% RSLogix 500 project 7.1.RSS, saved by version 8.30.00.16 %
PROJECT "UNTITLED"    % processor: Bul.1763 MicroLogix 1100 Series B %

PROGRAM FILES
  LAD 2   4 rungs

DATA FILES
  O0 OUTPUT  4 elements
  I1 INPUT  6 elements
  S2 STATUS  66 elements
  B3 BINARY  1 elements
  T4 TIMER  2 elements
  C5 COUNTER  1 elements
  R6 CONTROL  1 elements
  N7 INTEGER  1 elements
  F8 FLOAT  1 elements

LADDER 2
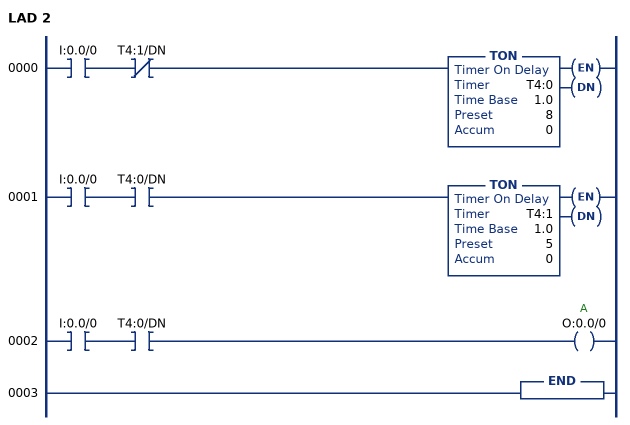
% Rung: 0 %
SOR XIC I:0.0/0 XIO T4:1/DN TON T4:0 1.0 8 0 EOR
% Rung: 1 %
SOR XIC I:0.0/0 XIC T4:0/DN TON T4:1 1.0 5 0 EOR
% Rung: 2 %
SOR XIC I:0.0/0 XIC T4:0/DN OTE O:0.0/0 EOR
%   O:0.0/0  "A" %
% Rung: 3 %
SOR END EOR

OTHER DOCUMENTED ADDRESSES
  O:0.0/1  "B"

DATA TABLE (non-zero values as saved)
DATA T4
% .PRE .ACC %
% T4:0 % 8 0
% T4:1 % 5 0
